// TIA Portal V21 export
TYPE "Std_Stazione"
   STRUCT
      IN : Struct
         SorgenteNonPronta : Bool;
         LivelloSorgenteInferiorePriorità : Bool;
         LivelloDestinazioneSuperiorePriorità : Bool;
         DestinazioneNonPronta : Bool;
         Feedback_Run : Bool;
      END_STRUCT;
      Hmi : Struct
         Abilita : Bool;
         Diagnostica : Struct
            StazioneAMonteNonPronta : Bool;   // La stazione a monta non è pronta ad inviare prodotto perciò non chiamo
            PrioritàLivelloDestinazione : Bool;   // Il tank di destinazione è salito sopra la priorità impostata per questa stazione
            PrioritàLivelloSorgente : Bool;   // Il tank di prelievo è sceso sotto la priorità impostata per questa stazione
            PercorsoNonAttivo : Bool;   // Il percorso è stato modificato ma non caricato
            DestinazioneNonPronta : Bool;   // La destinazione non è pronta a chiamare
            MancaAttivazioneDaHmi : Bool;   // Attivare con tasto ON OFF il percorso
            AttesaAdditivoPronto : Bool;   // La pompa mandata principale attende la pompa additivo
            AttesaPompaMandata : Bool;   // La pompa additivo attende la pompa mandata principale
            NessunaDestinazioneAttiva : Bool;   // Verifica di aver caricato la configurazione e di aver e di aver progettato il percorso correttamente
            TroppoPieno : Bool;   // Stazione serbatoio che ha raggiunto il livello massimo
            AttesaFeedbackRun : Bool;   // La stazione sta aspettando di vedere la chiamata a valle
         END_STRUCT;
      END_STRUCT;
      Prm : Struct
         ByPassChiamataDestinazione : Bool;   // Chiama sorgente anche se destinazione non chiama
         FeedbackRun : Struct
            Abilitazione : Bool;   // Se abilitato controlla l'ingresso di feedback
            ChiamaAncheDopoTimeot : Bool;   // Se scatta il timeout la stazione continua a tenere alta la chimata in uscita
            Attesa { S7_SetPoint := 'True'} : "Std_stTimer";
         END_STRUCT;
         AbilitazionePriorità : Struct   // Abilita se stabilire una prioità per le chiamate prodotto
            SugliArrivi : Bool;   // Abilitazione per chi manda prodotto verso di me
            SuEstrazioni : Bool;   // Abilitazione per chi estrae prodotto da me
         END_STRUCT;
         IgnoraDestinazione : Bool;
         FunzionamentoBatch : Bool;
      END_STRUCT;
      Allarmi : Struct
         Stato : Struct
            ConflittoMultiDest : Bool;
            AlmenoUnaDiagnosticaAttiva : Bool;
            TimeoutRun : Bool;
         END_STRUCT;
         EnWarnHmi : Struct
            ConflittoMultiDest : Bool;
            AlmenoUnaDiagnosticaAttiva : Bool;
            TimeoutRun : Bool;
         END_STRUCT;
         WordHMI : Word;
      END_STRUCT;
      Destinazione { S7_SetPoint := 'True'} : Array[0.."K_NumStazione"] of "Std_Stazioni";
      Dati : Struct
         RicezioneAdditivo : Struct   // Questa stazione funge da rifirimento per una stazione additiva
            Attiva : Bool;   // Indica che una stazione additiva è collegata a questa stazione
            K_StazioneRiferimento : Int;   // K stazione che si è collegata a me
         END_STRUCT;
         InvioAdditivo : Struct   // Questa stazione è una stazione di additivo (salamoia)
            Abilitazione : Bool;   // Abilita funzionamento additivo
            Attiva : Bool;   // Funzionamento additivo richiesto
            TuttiRiferimentiOk : Bool;   // Tutte le mandate sono pronte a chiamare
            K_StazioneRiferimento1 : Int;   // K stazione su cui fare riferimento per il calcolo additivo
            K_StazioneRiferimento2 : Int;   // K stazione2 per associare più sorgenti contemporanee
         END_STRUCT;
         DestAttivaPresente : Bool;
         K_StazioneDestinazione : Int;
         SorgAttivaPresente : Bool;   // Inidica che per la presente stazione almeno una sorgente progettata è attiva (Percorso attivo online)
         AlmenoUnaSorgenteProgettata : Bool;   // Inidica che per la presente stazione è progettata almeno una sorgente
         AlmenoUnaDestinazioneProgettata : Bool;   // Inidica che per la presente stazione è progettata almeno una destinazione
         IntMinLivelloTank_DaSorgente : Bool;
         IntMinLivelloTank_PerMotore : Bool;
         LivelloTank_DaSorgente : Real;   // Mi viene passato da una stazione serbatoio sorgente
         LivelloTank_PerMotore : Real;   // Dato per il motore di destinazione
         GestionePrioritàAttiva : Struct   // Indica che è presente una gestione priorità, perciò potrei essere fermato
            DaDestinazione : Bool;   // dalla stazione a cui mando prodoto
            DaSorgente : Bool;   // dalla stazione da cui ricevo prodoto
         END_STRUCT;
      END_STRUCT;
      OUT : Struct
         ProntaAChiamare : Bool;
         Chiamata : Bool;
      END_STRUCT;
      Rif_Inc : Struct
         K_Analogica : Int;
         K_Paratia : Int;
         K_Motore : Int;
         K_Pompa : Int;
         K_Stazione : Int;
      END_STRUCT;
   END_STRUCT;
   // // Destinazione[1] : Stazione M19
END_TYPE
